// TwinCAT 3 PLC project PLC1
// ProgramVersion: 3.1.4024.0
// libraries:
//   Tc2_Standard, * (Beckhoff Automation GmbH)
//   Tc2_System, * (Beckhoff Automation GmbH)
//   Tc3_Module, * (Beckhoff Automation GmbH)
// project tree:
//   GVLs/ GVL_ADS.TcGVL, GVL_IO.TcGVL
//   / PlcTask.TcTTO
//   POUs/FBs/ FB_WriteADS.TcPOU, FB_ReadADS.TcPOU
//   POUs/ MAIN.TcPOU
// real-time tasks:
//   TASK PlcTask: cycle T#10ms, priority 20, ADS port 350
// I/O:
//   DEVICE Device 1 (EtherCAT), AmsNetId 5.132.90.65.2.1
//     Term 1 (EK1200) [EK1200-7000 EtherCAT Power supply (1,5A E-Bus)]
//       Term 2 (EL6601) [EL6601 1 Port Switch (Ethernet, CoE)]
//       Term 3 (EL9011) [EL9011 End Terminal]
//   DEVICE Device 2 (NOV-DP-RAM)
//   DEVICE Device 3 (CX7000), AmsNetId 5.132.90.65.4.1
//     Term 1 (CX7028) [CX7028-0000-0118]
//       modules: Module 1 (DIO_2x), Module 3 (DIO_2x), Module 5 (DI_2x), Module 7 (DI_2x)
//   DEVICE Device 4 (COM Port)
//   DEVICE Device 5 (COM Port)
// variable links:
//   PLC1/PLC1 Instance <-> Device 1 (EtherCAT)
//     PlcTask Inputs/GVL_IO.uiMasterState <-> Inputs/DevState
//   PLC1/PLC1 Instance <-> Device 3 (CX7000)/Term 1 (CX7028)
//     PlcTask Inputs/GVL_IO.bInput1 <-> Module 1 (DIO_2x)/DIO_2x Inputs Channel 1/Input

CONFIGURATION PLC1
    RESOURCE PLC ON TwinCAT3
        TASK PlcTask(INTERVAL := T#10ms, PRIORITY := 20);
        PROGRAM MAIN WITH PlcTask : MAIN;
    END_RESOURCE
END_CONFIGURATION

// ---- GVLs/GVL_ADS.TcGVL
{attribute 'Tc2GvlVarNames'}
VAR_GLOBAL
	Array_LPB_TDA_INT AT%MB1000: ARRAY[0..20] OF INT;
	Array_INT_Test : ARRAY [0..20] OF INT;
END_VAR

// ---- GVLs/GVL_IO.TcGVL
{attribute 'qualified_only'}
VAR_GLOBAL
	bInput1 AT%I* : BOOL;
	uiMasterState AT%I* : UINT;
END_VAR

// ---- POUs/MAIN.TcPOU
PROGRAM MAIN
VAR
	fbReadADS_1		: FB_ReadADS;
	bStart			: BOOL;
	bReset			: BOOL;
	fbWriteADS_1	: FB_WriteADS;
	bStartWrite		: BOOL;
	bResetWrite		: BOOL;
	i				: INT;
END_VAR

actComunicacao();

FOR i := 0 TO 20 DO
	GVL_ADS.Array_INT_Test[i] := i*33;
END_FOR

ACTION actComunicacao:
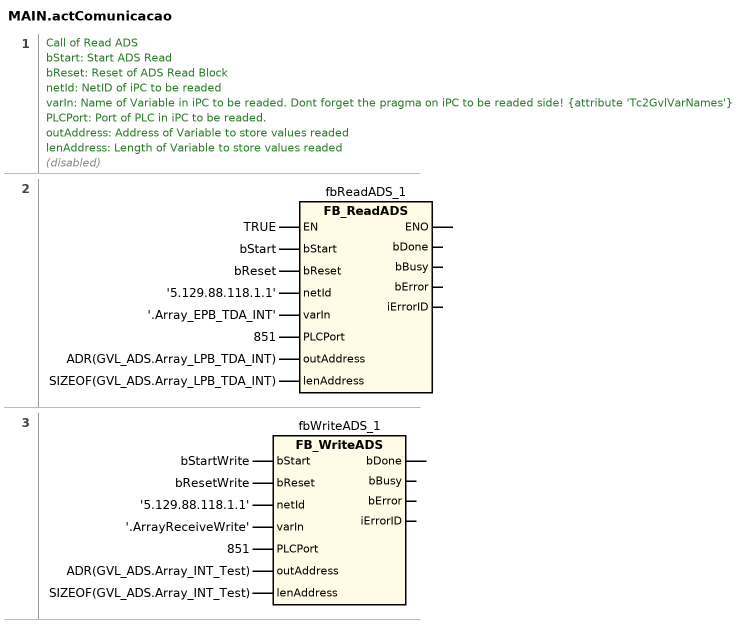
// NETWORK 1 (disabled)
// Call of Read ADS
// bStart: Start ADS Read
// bReset: Reset of ADS Read Block
// netId: NetID of iPC to be readed
// varIn: Name of Variable in iPC to be readed. Dont forget the pragma on iPC to be readed side! {attribute 'Tc2GvlVarNames'}
// PLCPort: Port of PLC in iPC to be readed.
// outAddress: Address of Variable to store values readed
// lenAddress: Length of Variable to store values readed

// NETWORK 2
fbReadADS_1(
    bStart := bStart,
    bReset := bReset,
    netId := '5.129.88.118.1.1',
    varIn := '.Array_EPB_TDA_INT',
    PLCPort := 851,
    outAddress := ADR(GVL_ADS.Array_LPB_TDA_INT),
    lenAddress := SIZEOF(GVL_ADS.Array_LPB_TDA_INT)); // FB_ReadADS

// NETWORK 3
fbWriteADS_1(
    bStart := bStartWrite,
    bReset := bResetWrite,
    netId := '5.129.88.118.1.1',
    varIn := '.ArrayReceiveWrite',
    PLCPort := 851,
    outAddress := ADR(GVL_ADS.Array_INT_Test),
    lenAddress := SIZEOF(GVL_ADS.Array_INT_Test)); // FB_WriteADS
END_ACTION

END_PROGRAM

// ---- POUs/FBs/FB_ReadADS.TcPOU
FUNCTION_BLOCK FB_ReadADS
(* Recomendada a leitura de arrays para melhor performance *)
VAR_INPUT
	bStart			: BOOL; // Start Comm	
	bReset			: BOOL;
	netId 			: T_AmsNetId;
	varIn 			: STRING;
	PLCPort			: UINT;
	outAddress		: DWORD;
	lenAddress		: UDINT;	
END_VAR         	
VAR_OUTPUT      		
	bDone 			: BOOL;
	bBusy 			: BOOL;
	bError 			: BOOL;
	iErrorID 		: UDINT;
END_VAR
VAR
	netidAux 		: T_AmsNetId;     	          	
	getHandle 		: ADSRDWRT; (*Bloco para obter o handle*)
	handles 		: UDINT; (*Handle para a variavel remota*)
	reader 			: ADSREAD; (*Bloco de leitura via ADS*)  
	state 			: INT;
	varAux			: STRING;
	iHandleErrorId	: UDINT;
	iReadErrorId	: UDINT;
	iConsecutiveError		: INT; (* Erros consecutivos *)
	TON_ConsecutiveError	: TON;
	TON_ReadOK		: TON;
END_VAR

IF bReset THEN
	state := 0;
	iConsecutiveError := 0;
END_IF

CASE state OF
	0: // Start of ADS Communication
		bDone := FALSE;
		iErrorID := 0;
		netidAux 	:= netid;		
		varAux 		:= varIn;
			
		bBusy	 	:= FALSE; // Status Variable to Inform User
		bError		:= FALSE; // Status Variable to Inform User
		
		getHandle(WRTRD:= FALSE);
		reader(READ:= FALSE);
		
		IF NOT bReset AND bStart THEN			
			state 		:= 10;	
		END_IF
		
	10: // ADS get Handler
		getHandle(
			NETID		:= netidAux,
			PORT		:= PLCPort,
			IDXGRP		:= 16#F003,
			IDXOFFS		:= 0,
			WRITELEN	:= INT_TO_UDINT(LEN(varAux)+1),
			READLEN		:= SIZEOF(handles),
			SRCADDR		:= ADR(varAux),
			DESTADDR	:= ADR(handles),
			WRTRD		:= TRUE,
			TMOUT		:= T#10S,
			BUSY 		=> ,
			ERR 		=> ,
			ERRID 		=>
		);
		IF NOT getHandle.BUSY THEN
			IF getHandle.ERR THEN				
				iHandleErrorId := getHandle.ERRID;			
				state := 999;
			ELSE
				state := 20;
			END_IF
		END_IF
		
	20:	// ADS Read 
		reader(
			NETID			:= netidAux,
			PORT			:= PLCPort,
			IDXGRP			:= 16#F005,
			IDXOFFS			:= handles,
			LEN				:= lenAddress,
			DESTADDR		:= outAddress,
			READ			:= TRUE,
			TMOUT			:= T#10S,
			BUSY 			=>,
			ERR 			=>,
			ERRID 			=>
		);
		
		IF NOT reader.BUSY THEN 
			IF reader.ERR THEN
				iReadErrorId := reader.ERRID;			
				state := 999;
			ELSE			
				state := 30;
			END_IF				
		END_IF
		
	30: (* Close Open Handles *)
		iConsecutiveError := 0;		
		getHandle(
			NETID		:= netidAux,
			PORT		:= PLCPort,
			IDXGRP		:= 16#F006,
			IDXOFFS		:= 0,
			WRITELEN	:= INT_TO_UDINT(LEN(varAux)+1),
			READLEN		:= SIZEOF(handles),
			SRCADDR		:= ADR(varAux),
			DESTADDR	:= ADR(handles),
			WRTRD		:= TRUE,
			TMOUT		:= T#10S,
			BUSY 		=> ,
			ERR 		=> ,
			ERRID 		=>
		);
		IF NOT getHandle.BUSY THEN
			IF getHandle.ERR THEN
				iHandleErrorId := getHandle.ERRID;
				state := 999;
			ELSE				
				state := 40;
			END_IF
		END_IF
		
	40: // Wait until next read
		IF TON_ReadOK.Q THEN
			bDone := TRUE;
			state := 0;
		END_IF
		
	999: // Error State	
		IF iConsecutiveError > 3 THEN	
			bError		:= TRUE; // Status Variable to Inform User
			iErrorID	:= iReadErrorId OR iHandleErrorId;
			
			getHandle(WRTRD:= FALSE);
			reader(READ:= FALSE);
		ELSE
			iConsecutiveError := iConsecutiveError + 1;
			IF TON_ConsecutiveError.Q THEN
				state := 0;
			END_IF						
		END_IF
END_CASE

TON_ReadOK(IN:= state=40, PT:= T#500MS, Q=> , ET=> );	
TON_ConsecutiveError(IN:= state=999, PT:= T#2S, Q=> , ET=> );


bBusy := state > 0 AND state < 999; // Status Variable to Inform User

END_FUNCTION_BLOCK

// ---- POUs/FBs/FB_WriteADS.TcPOU
FUNCTION_BLOCK FB_WriteADS
(* Recomendada a leitura de arrays para melhor performance *)
VAR_INPUT
	bStart			: BOOL; // Start Comm	
	bReset			: BOOL;
	netId 			: T_AmsNetId;
	varIn 			: STRING;
	PLCPort			: UINT;
	outAddress		: DWORD;
	lenAddress		: UDINT;	
END_VAR         	
VAR_OUTPUT      		
	bDone 			: BOOL;
	bBusy 			: BOOL;
	bError 			: BOOL;
	iErrorID 		: UDINT;
END_VAR
VAR
	netidAux 		: T_AmsNetId;     	          	
	getHandle 		: ADSRDWRT; (*Bloco para obter o handle*)
	handles 		: UDINT; (*Handle para a variavel remota*)
	writer 			: ADSWRITE; (*Bloco de leitura via ADS*)  
	state 			: INT;
	varAux			: STRING;
	iHandleErrorId	: UDINT;
	iWriteErrorId	: UDINT;
	iConsecutiveError		: INT; (* Erros consecutivos *)
	TON_ConsecutiveError	: TON;
	TON_ReadOK		: TON;
END_VAR

IF bReset THEN
	state := 0;
	iConsecutiveError := 0;
END_IF

CASE state OF
	0: // Start of ADS Communication
		bDone := FALSE;
		iErrorID := 0;
		netidAux 	:= netid;		
		varAux 		:= varIn;
			
		bBusy	 	:= FALSE; // Status Variable to Inform User
		bError		:= FALSE; // Status Variable to Inform User
		
		getHandle(WRTRD:= FALSE);
		writer(WRITE:= FALSE);
		
		IF NOT bReset AND bStart THEN			
			state 		:= 10;	
		END_IF
		
	10: // ADS get Handler
		getHandle(
			NETID		:= netidAux,
			PORT		:= PLCPort,
			IDXGRP		:= 16#F003,
			IDXOFFS		:= 0,
			WRITELEN	:= INT_TO_UDINT(LEN(varAux)+1),
			READLEN		:= SIZEOF(handles),
			SRCADDR		:= ADR(varAux),
			DESTADDR	:= ADR(handles),
			WRTRD		:= TRUE,
			TMOUT		:= T#10S,
			BUSY 		=> ,
			ERR 		=> ,
			ERRID 		=>
		);
		IF NOT getHandle.BUSY THEN
			IF getHandle.ERR THEN				
				iHandleErrorId := getHandle.ERRID;			
				state := 999;
			ELSE
				state := 20;
			END_IF
		END_IF
		
	20:	// ADS Read 
		writer(
			NETID:= netidAux, 
			PORT:= PLCPort, 
			IDXGRP:= 16#F005, 
			IDXOFFS:= handles, 
			LEN:= lenAddress, 
			SRCADDR:= outAddress, 
			WRITE:= TRUE, 
			TMOUT:= T#10S, 
			BUSY=> , 
			ERR=> , 
			ERRID=> 
		);
		
		IF NOT writer.BUSY THEN 
			IF writer.ERR THEN
				iWriteErrorId := writer.ERRID;			
				state := 999;
			ELSE			
				state := 30;
			END_IF				
		END_IF
		
	30: (* Close Open Handles *)
		iConsecutiveError := 0;		
		getHandle(
			NETID		:= netidAux,
			PORT		:= PLCPort,
			IDXGRP		:= 16#F006,
			IDXOFFS		:= 0,
			WRITELEN	:= INT_TO_UDINT(LEN(varAux)+1),
			READLEN		:= SIZEOF(handles),
			SRCADDR		:= ADR(varAux),
			DESTADDR	:= ADR(handles),
			WRTRD		:= TRUE,
			TMOUT		:= T#10S,
			BUSY 		=> ,
			ERR 		=> ,
			ERRID 		=>
		);
		IF NOT getHandle.BUSY THEN
			IF getHandle.ERR THEN
				iHandleErrorId := getHandle.ERRID;
				state := 999;
			ELSE				
				state := 40;
			END_IF
		END_IF
		
	40: // Wait until next read
		IF TON_ReadOK.Q THEN
			bDone := TRUE;
			state := 0;
		END_IF
		
	999: // Error State	
		IF iConsecutiveError > 3 THEN	
			bError		:= TRUE; // Status Variable to Inform User
			iErrorID	:= iWriteErrorId OR iHandleErrorId;
			
			getHandle(WRTRD:= FALSE);
			writer(WRITE:= FALSE);
		ELSE
			iConsecutiveError := iConsecutiveError + 1;
			IF TON_ConsecutiveError.Q THEN
				state := 0;
			END_IF						
		END_IF
END_CASE

TON_ReadOK(IN:= state=40, PT:= T#500MS, Q=> , ET=> );	
TON_ConsecutiveError(IN:= state=999, PT:= T#2S, Q=> , ET=> );


bBusy := state > 0 AND state < 999; // Status Variable to Inform User

END_FUNCTION_BLOCK
